// TIA Portal V17 export
// export: Created 2025-04-14T03:01:51.0590205Z, ExportSetting WithDefaults, DisplayName Totally Integrated Automation Portal, DisplayVersion V17, DisplayName TIA Portal Openness, DisplayVersion V17, DisplayName TIA Portal Version Control Interface, DisplayVersion V17, DisplayName SINAMICS Startdrive Advanced, DisplayVersion V17, DisplayName SINAMICS Startdrive G130, G150, S120, S150, SINAMICS MV, S210, DisplayVersion V17, DisplayName SINAMICS Startdrive G110M, G120, G120C, G120D, G120P, G115D, DisplayVersion V17, DisplayName STEP 7 Professional, DisplayVersion V17, DisplayName STEP 7 Safety, DisplayVersion V17, DisplayName WinCC Advanced, DisplayVersion V17
TYPE "UDT_Valve_Map"
// stored: IsFailsafeCompliant false
   STRUCT
      IN_xOpenFeedback : Bool;   // 传感器开
      IN_xCloseFeedback : Bool;   // 传感器关
      OUT_xActualOut : Bool;   // 阀门控制
   END_STRUCT;
END_TYPE
